(* CODESYS project testrepo

Project tree, tasks and I/O mapping:
  Device : HY-TTC 510, TTControl, order no. n/a, version 1.8.0.0
    application Application
      libraries: lib500, 1.8.0.0 (TTControl); lib500_types, 1.8.0.0 (TTControl); lib500_syscom, 1.8.0.0 (TTControl); Standard, 3.5.18.0 (System); Test Manager IEC Unit Test, 5.1.0.0 (Intern)
      task _ErrorCallback (externalevent, external event ErrorCallback, priority 1) calls _ErrorCB_PRG
      task _NotificationCallback (externalevent, external event NotificationCallback, priority 0) calls _NotificationCB_PRG
      task MainTask (cyclic, interval t#10ms, priority 2, watchdog t#10ms x 1) calls PLC_PRG
      program _ErrorCB_PRG [ST]
      program _NotificationCB_PRG [ST]
      function funkcja [ST]
      global variables GVL
      program PLC_PRG [ST]
    CANs : CANs, TTControl, order no. n/a, version 1.8.0.0
      CAN0 : CAN0, TTControl, order no. n/a, version 1.8.0.0
      CAN1 : CAN1, TTControl, order no. n/a, version 1.8.0.0
      CAN2 : CAN2, TTControl, order no. n/a, version 1.8.0.0
    System : System, TTControl, order no. n/a, version 1.8.0.0
        unmapped channels: mode, error, mode, error, mode, error, mode, error, mode, error, mode, error, shutdown, error, enable_error_group_0, enable_error_group_1, diag_status, safe_state, error, driver_init_error, UBAT, Terminal_15, WakeUp, Temperature, SSW0, SSW1, SSUP0, SSUP1, SSUP2, status, write, boot_error, trigger_error, Powerstage, SSW0, SSW1, SSUP0, SSUP1, SSUP2, Terminal_15,
          WakeUp, ExtShutOff0, ExtShutOff1
      Analog_Inputs_2Mode_10V : AIN_2Mode_10V, TTControl, order no. n/a, version 1.8.0.0
        Pin 107
          <Empty>
        Pin 108
          <Empty>
        Pin 109
          <Empty>
        Pin 110
          <Empty>
        Pin 131
          <Empty>
        Pin 132
          <Empty>
        Pin 133
          <Empty>
        Pin 134
          <Empty>
      Analog_Inputs_2Mode_32V : AIN_2Mode_32V, TTControl, order no. n/a, version 1.8.0.0
        Pin 111
          <Empty>
        Pin 112
          <Empty>
        Pin 113
          <Empty>
        Pin 114
          <Empty>
        Pin 135
          <Empty>
        Pin 136
          <Empty>
        Pin 137
          <Empty>
        Pin 138
          <Empty>
      Analog_Inputs_3Mode : AIN_3Mode, TTControl, order no. n/a, version 1.8.0.0
        Pin 103
          <Empty>
        Pin 104
          <Empty>
        Pin 105
          <Empty>
        Pin 106
          <Empty>
        Pin 127
          <Empty>
        Pin 128
          <Empty>
        Pin 129
          <Empty>
        Pin 130
          <Empty>
      Digital_Inputs : DIN, TTControl, order no. n/a, version 1.8.0.0
        Pin 101
          <Empty>
        Pin 102
          <Empty>
        Pin 125
          <Empty>
        Pin 126
          <Empty>
        Pin 150
          <Empty>
        Pin 151
          <Empty>
        Pin 174
          <Empty>
        Pin 175
          <Empty>
      Digital_Outputs_HS : HSDOUT, TTControl, order no. n/a, version 1.8.0.0
        Pin 149
          <Empty>
        Pin 152
          <Empty>
        Pin 155
          <Empty>
        Pin 158
          <Empty>
        Pin 173
          <Empty>
        Pin 176
          <Empty>
        Pin 179
          <Empty>
        Pin 182
          <Empty>
      Digital_Outputs_LS : LSDOUT, TTControl, order no. n/a, version 1.8.0.0
        Pin 238
          <Empty>
        Pin 239
          <Empty>
        Pin 240
          <Empty>
        Pin 241
          <Empty>
        Pin 251
          <Empty>
        Pin 252
          <Empty>
        Pin 253
          <Empty>
        Pin 254
          <Empty>
      PVG_Outputs : PVG, TTControl, order no. n/a, version 1.8.0.0
        Pin 161
          <Empty>
        Pin 164
          <Empty>
        Pin 167
          <Empty>
        Pin 170
          <Empty>
        Pin 185
          <Empty>
        Pin 188
          <Empty>
        Pin 191
          <Empty>
        Pin 194
          <Empty>
      PWM_Outputs : PWM, TTControl, order no. n/a, version 1.8.0.0
        Safety_switch_0 : PWM_SSW0, TTControl, order no. n/a, version 1.8.0.0
          Pin 153
            <Empty>
          Pin 156
            <Empty>
          Pin 159
            <Empty>
          Pin 162
            <Empty>
          Pin 177
            <Empty>
          Pin 180
            <Empty>
          Pin 183
            <Empty>
          Pin 186
            <Empty>
        Safety_switch_1 : PWM_SSW1, TTControl, order no. n/a, version 1.8.0.0
          Pin 154
            <Empty>
          Pin 157
            <Empty>
          Pin 160
            <Empty>
          Pin 163
            <Empty>
          Pin 178
            <Empty>
          Pin 181
            <Empty>
          Pin 184
            <Empty>
          Pin 187
            <Empty>
      Timer_Inputs : TIN, TTControl, order no. n/a, version 1.8.0.0
        Pin 122
          <Empty>
        Pin 123
          <Empty>
        Pin 124
          <Empty>
        Pin 146
          <Empty>
        Pin 147
          <Empty>
        Pin 148
          <Empty>
      Timer_Inputs_Cur : TIN_Cur, TTControl, order no. n/a, version 1.8.0.0
        Pin 115
          <Empty>
        Pin 116
          <Empty>
        Pin 117
          <Empty>
        Pin 139
          <Empty>
        Pin 140
          <Empty>
        Pin 141
          <Empty>
*)

// Device/Application/GVL
{attribute 'qualified_only'}
VAR_GLOBAL
END_VAR

// Device/Application/_ErrorCB_PRG
PROGRAM _ErrorCB_PRG
VAR
	diag_state : lib500_types.DIAG_STATETYPE := lib500_types.DIAG_STATETYPE.DIAG_STATE_DISABLED;
	watchdog_state : lib500_types.DIAG_WD_STATETYPE := lib500_types.DIAG_WD_STATETYPE.DIAG_WD_STATE_UNKNOWN;
	error : lib500_types.DIAG_ERRORCODE := (error_code := lib500_types.DIAG_ERRORTYPE.DIAG_E_NOERROR, 
                                            device_num := lib500_types.DIAG_DEVICETYPE.DIAG_DEV_NONE,
                                            faulty_value := 0);
	return_code : lib500_types.IO_ERRORTYPE := lib500_types.IO_ERRORTYPE.IO_E_UNKNOWN;
	
	reaction : lib500_types.DIAG_REACTION := lib500_types.DIAG_REACTION.DIAG_ERR_SAFESTATE;
	
	call_count : UDINT := 0;
END_VAR

(* get the reason for the error callback *)
return_code := lib500.DIAG_CDS_GetErrorReason(ADR(diag_state), 
                                              ADR(watchdog_state),
                                              ADR(error));

(* custom handler code can be placed here *)

(* the choices for the reactions are:
   -> lib500_types.DIAG_REACTION.DIAG_ERR_NOACTION
   -> lib500_types.DIAG_REACTION.DIAG_ERR_SAFESTATE
   -> lib500_types.DIAG_REACTION.DIAG_ERR_DISABLE_SSW0
   -> lib500_types.DIAG_REACTION.DIAG_ERR_DISABLE_SSW1
   -> lib500_types.DIAG_REACTION.DIAG_ERR_DISABLE_HS00
   -> lib500_types.DIAG_REACTION.DIAG_ERR_DISABLE_HS01
   -> lib500_types.DIAG_REACTION.DIAG_ERR_DISABLE_HS02
   -> lib500_types.DIAG_REACTION.DIAG_ERR_DISABLE_HS03
   -> lib500_types.DIAG_REACTION.DIAG_ERR_DISABLE_HS04
   -> lib500_types.DIAG_REACTION.DIAG_ERR_DISABLE_HS05
   -> lib500_types.DIAG_REACTION.DIAG_ERR_DISABLE_HS06
   -> lib500_types.DIAG_REACTION.DIAG_ERR_DISABLE_HS07
   
   it's also possible to combine (binary-or) reactions, like:
   -> lib500_types.DIAG_REACTION.DIAG_ERR_DISABLE_SSW0 OR 
      lib500_types.DIAG_REACTION.DIAG_ERR_DISABLE_SSW1
*)

(* pass the error reaction to the DIAG system *)
lib500.DIAG_CDS_SetErrorReaction(reaction);

(* increment call count *)
call_count := call_count + 1;

END_PROGRAM

// Device/Application/_NotificationCB_PRG
PROGRAM _NotificationCB_PRG
VAR
	diag_state : lib500_types.DIAG_STATETYPE := lib500_types.DIAG_STATETYPE.DIAG_STATE_DISABLED;
	watchdog_state : lib500_types.DIAG_WD_STATETYPE := lib500_types.DIAG_WD_STATETYPE.DIAG_WD_STATE_UNKNOWN;
	error : lib500_types.DIAG_ERRORCODE := (error_code := lib500_types.DIAG_ERRORTYPE.DIAG_E_NOERROR, 
                                            device_num := lib500_types.DIAG_DEVICETYPE.DIAG_DEV_NONE,
                                            faulty_value := 0);
	return_code : lib500_types.IO_ERRORTYPE := lib500_types.IO_ERRORTYPE.IO_E_UNKNOWN;
	
	call_count : UDINT := 0;
END_VAR

(* get the reason for the notification callback *)
return_code := lib500.DIAG_CDS_GetNotificationReason(ADR(diag_state), 
                                                     ADR(watchdog_state),
                                                     ADR(error));

(* custom handler code can be placed here *)

(* increment call count *)
call_count := call_count + 1;

END_PROGRAM

// Device/Application/PLC_PRG
PROGRAM PLC_PRG
VAR
	testowy_git:INT;
END_VAR

testowy_git:=testowy_git+2;

END_PROGRAM

// Device/Application/funkcja
FUNCTION funkcja : bool
VAR_INPUT
END_VAR
VAR
END_VAR

END_FUNCTION
